(* IEC 61131-3 sources: repolevel_ST_code_completion/output/0127完整版本_带planner/repoeval_open-type_dual-axis_winding_machine/readful_result_no_provide, 5 files *)

(* ---- F_CalculateRadius.st ---- *)
FUNCTION F_CalculateRadius : LREAL
VAR_INPUT
  lD : LREAL;             // 两轴中心距离
  lHold : LREAL;          // 测量开始时的AxisV位置
  lHnew : LREAL;          // 测量结束时的AxisV位置
  lTk : LREAL;            // 材料厚度
  lOffset : LREAL;        // 高度偏移量
END_VAR
VAR
  lDeltaH : LREAL;          // 轴位置变化量
  lEffectiveHeight : LREAL; // 总的有效高度
  lRadius : LREAL;          // 计算得到的半径值
END_VAR

// 计算轴位置变化量
lDeltaH := ABS(lHnew - lHold);

// 计算总的有效高度
lEffectiveHeight := lDeltaH + lTk + lOffset;

// 根据两轴中心距离和有效高度计算半径
lRadius := SQRT(EXPT(lD / 2, 2) + EXPT(lEffectiveHeight, 2));

// 返回计算得到的半径值
F_CalculateRadius := lRadius;
RETURN;
END_FUNCTION

(* ---- CheckF.st ---- *)
VAR
END_VAR

IF lH <> 0 THEN
    lF := 9.8 * lM / (2 * COS(ATAN(lL / lH)));
ELSE
    lF := 0;
END_IF;
END_FUNCTION_BLOCK

(* ---- F_CompensateVelocity.st ---- *)
VAR
    lDeltaPos       : LREAL;    // 位置变化量
    lDeltaRadius    : LREAL;    // 半径变化量
    lCompFactor     : LREAL;    // 速度补偿系数
    lAdjustedRadius : LREAL;    // 调整后的半径
END_VAR

// 1. 计算位置变化量
lDeltaPos := lNewPos - lOldPos;

// 2. 判断运动方向并校正位置变化量
IF lDeltaPos = 0 THEN
    lDeltaPos := 0; // 保持不变
ELSIF lDeltaPos < 0 THEN
    lDeltaPos := -ABS(lDeltaPos); // 确保方向正确
ELSE
    lDeltaPos := ABS(lDeltaPos);
END_IF

// 3. 计算半径变化量
lDeltaRadius := lDeltaPos * lTk;

// 4. 根据放卷或收卷逻辑调整半径
IF bUnwinding THEN
    lAdjustedRadius := lRadius - lDeltaRadius; // 放卷：半径减小
ELSE
    lAdjustedRadius := lRadius + lDeltaRadius; // 收卷：半径增加
END_IF

// 避免半径过小导致除零错误
IF lAdjustedRadius < 0.01 THEN
    lAdjustedRadius := 0.01;
END_IF

// 5. 计算速度补偿系数
lCompFactor := lRadius / lAdjustedRadius;

// 6. 使用补偿系数调整速度
F_CompensateVelocity := lCurrentVel * lCompFactor;
RETURN;
END_FUNCTION

(* ---- SeekHome.st ---- *)
VAR
	_nState		:	USINT;
	_fbMoveVel	:	MC_MoveVelocity;
	_fbMoveAbs	:	MC_MoveAbsolute;
	_fbHalt		:	MC_Halt;
	_fbSetPos	:	MC_SetPosition;
	_fbRtrig	:	R_TRIG;
	_fbFtrig	:	F_TRIG;
	_nBDirection	:	MC_DIRECTION;
	_fTempPos		:	LREAL;
	_xHomeActive	:	BOOL;
	_xAbortActive	:	BOOL;
END_VAR

IF _xHome THEN
	_xHomeActive := TRUE;
	_xAbortActive := FALSE;
	_xBusy := TRUE;
	_xDone := FALSE;
	_xErr := FALSE;
	_iErrId := 0;
	_nState := 1;
ELSIF _xAbort THEN
	_xAbortActive := TRUE;
	_xHomeActive := FALSE;
	_xBusy := FALSE;
	_xDone := FALSE;
	_xErr := FALSE;
	_iErrId := 0;
	_nState := 0;
END_IF

CASE _nState OF
	0: // Idle state
		IF _xAbortActive THEN
			_fbHalt.Execute := TRUE;
			_fbHalt.Axis := _Axis;
			_fbHalt.Deceleration := _fHomeDec;
			_fbHalt.Execute := FALSE;
			_xAbortActive := FALSE;
		END_IF

	1: // Start homing
		IF _xHomeActive THEN
			_fbMoveVel.Execute := TRUE;
			_fbMoveVel.Axis := _Axis;
			_fbMoveVel.Velocity := _fFastHomeVel;
			_fbMoveVel.Acceleration := _fHomeAcc;
			_fbMoveVel.Deceleration := _fHomeDec;
			_fbMoveVel.Direction := _nDirection;
			IF _fbMoveVel.Done THEN
				_fbMoveVel.Execute := FALSE;
				_nState := 2;
			END_IF
		END_IF

	2: // Monitor reference switch
		IF _xReferenceSwitch THEN
			_fbMoveVel.Execute := FALSE;
			_fbMoveAbs.Execute := TRUE;
			_fbMoveAbs.Axis := _Axis;
			_fbMoveAbs.Position := _fHomePos;
			_fbMoveAbs.Velocity := _fSlowHomeVel;
			_fbMoveAbs.Acceleration := _fHomeAcc;
			_fbMoveAbs.Deceleration := _fHomeDec;
			IF _fbMoveAbs.Done THEN
				_fbMoveAbs.Execute := FALSE;
				_nState := 3;
			END_IF
		END_IF

	3: // Monitor index pulse
		IF _xIndexPulse THEN
			_fbSetPos.Execute := TRUE;
			_fbSetPos.Axis := _Axis;
			_fbSetPos.Position := 0.0;
			IF _fbSetPos.Done THEN
				_fbSetPos.Execute := FALSE;
				_xDone := TRUE;
				_xBusy := FALSE;
				_nState := 0;
			END_IF
		END_IF

	ELSE
		_xErr := TRUE;
		_iErrId := 1; // Unknown state error
		_xBusy := FALSE;
		_nState := 0;
END_CASE
END_FUNCTION_BLOCK

(* ---- StaDisplay.st ---- *)
VAR
END_VAR

CASE iStatus OF
    0:
        Y1 := FALSE;
        Y2 := FALSE;
        Y3 := FALSE;
        Y4 := FALSE;
        Y5 := FALSE;
        Y6 := FALSE;
    1:
        Y1 := TRUE;
        Y2 := FALSE;
        Y3 := FALSE;
        Y4 := FALSE;
        Y5 := FALSE;
        Y6 := FALSE;
    2:
        Y1 := FALSE;
        Y2 := TRUE;
        Y3 := FALSE;
        Y4 := FALSE;
        Y5 := FALSE;
        Y6 := FALSE;
    3:
        Y1 := FALSE;
        Y2 := FALSE;
        Y3 := TRUE;
        Y4 := FALSE;
        Y5 := FALSE;
        Y6 := FALSE;
    4:
        Y1 := FALSE;
        Y2 := FALSE;
        Y3 := FALSE;
        Y4 := TRUE;
        Y5 := FALSE;
        Y6 := FALSE;
    5:
        Y1 := FALSE;
        Y2 := FALSE;
        Y3 := FALSE;
        Y4 := FALSE;
        Y5 := TRUE;
        Y6 := FALSE;
    6:
        Y1 := FALSE;
        Y2 := FALSE;
        Y3 := FALSE;
        Y4 := FALSE;
        Y5 := FALSE;
        Y6 := TRUE;
    ELSE
        Y1 := FALSE;
        Y2 := FALSE;
        Y3 := FALSE;
        Y4 := FALSE;
        Y5 := FALSE;
        Y6 := FALSE;
END_CASE;
END_FUNCTION_BLOCK
